(* Logix 5000 project; controller ODSI_Testing vendor 1 type 14 code 151 rev 20.19; software revision 20.05 *)

TASK MainTask (continuous, watchdog 500 ms) : MainProgram

MODULES
   Local : vendor 1 type 14 code 151 (Compact 0, rev 20.19)
      Expansion_Input_1 : 1769-IQ16 (Compact 4, rev 1.1, Input RPI 20 ms)   // Sink or Source
      Expansion_Input_2 : 1769-IQ32 (Compact 6, rev 3.1, Input RPI 20 ms)
      Discrete_IO : Embedded (Compact 1, rev 3.1, Output RPI 20 ms)
      Analog_IO : Embedded (Compact 2, rev 1.1, Output RPI 80 ms)
      Counters : Embedded (Compact 3, rev 1.1, Output RPI 20 ms)
      Expansion_Output_1 : vendor 1 type 7 code 75 (Compact 5, rev 1.1, Output RPI 20 ms)
END_MODULES

VAR_GLOBAL   (* controller tags *)
   B11_DELAY_ONS : BOOL;
   B12_DELAY_ONS : BOOL;
   B1_DELAY_ONS : BOOL;
   B9_DELAY_ONS : BOOL;
   DutyCycleOutput : BOOL := 1;   // 1.25 second duty cycle output
   DutyCycleTimer : TIMER := (PRE := 2500, ACC := 2111, EN := 1, TT := 1);   // Accumulates preset time then resets
   HMI_Stop_B1 : BOOL;   // Stop PB on HMI
   HMI_Stop_B11 : BOOL;   // Stop PB on HMI
   HMI_Stop_B12 : BOOL;   // Stop PB on HMI
   HMI_Stop_B9 : BOOL;   // Stop PB on HMI
   ODSI_Fail_Sample1_B1 : ALIAS FOR Local:4:I.Data.8;   // ODSI sent a fail signal for sample 1
   ODSI_Fail_Sample1_B11 : ALIAS FOR Local:1:I.Data.8;   // ODSI sent a fail signal for sample 1
   ODSI_Fail_Sample1_B12 : ALIAS FOR Local:6:I.Data.24;   // ODSI sent a fail signal for sample 1
   ODSI_Fail_Sample1_B9 : ALIAS FOR Local:6:I.Data.8;   // ODSI sent a fail signal for sample 1
   ODSI_Fail_Sample2_B1 : ALIAS FOR Local:4:I.Data.10;   // ODSI sent a fail signal for sample 2
   ODSI_Fail_Sample2_B11 : ALIAS FOR Local:1:I.Data.10;   // ODSI sent a fail signal for sample 2
   ODSI_Fail_Sample2_B12 : ALIAS FOR Local:6:I.Data.26;   // ODSI sent a fail signal for sample 2
   ODSI_Fail_Sample2_B9 : ALIAS FOR Local:6:I.Data.10;   // ODSI sent a fail signal for sample 2
   ODSI_Fail_Sample3_B1 : ALIAS FOR Local:4:I.Data.12;   // ODSI sent a fail signal for sample 3
   ODSI_Fail_Sample3_B11 : ALIAS FOR Local:1:I.Data.12;   // ODSI sent a fail signal for sample 3
   ODSI_Fail_Sample3_B12 : ALIAS FOR Local:6:I.Data.28;   // ODSI sent a fail signal for sample 3
   ODSI_Fail_Sample3_B9 : ALIAS FOR Local:6:I.Data.12;   // ODSI sent a fail signal for sample 3
   ODSI_Pass_Sample1_B1 : ALIAS FOR Local:4:I.Data.7;   // ODSI sent a pass signal for sample 1
   ODSI_Pass_Sample1_B11 : ALIAS FOR Local:1:I.Data.7;   // ODSI sent a pass signal for sample 1
   ODSI_Pass_Sample1_B12 : ALIAS FOR Local:6:I.Data.23;   // ODSI sent a pass signal for sample 1
   ODSI_Pass_Sample1_B9 : ALIAS FOR Local:6:I.Data.7;   // ODSI sent a pass signal for sample 1
   ODSI_Pass_Sample2_B1 : ALIAS FOR Local:4:I.Data.9;   // ODSI sent a pass signal for sample 2
   ODSI_Pass_Sample2_B11 : ALIAS FOR Local:1:I.Data.9;   // ODSI sent a pass signal for sample 2
   ODSI_Pass_Sample2_B12 : ALIAS FOR Local:6:I.Data.25;   // ODSI sent a pass signal for sample 2
   ODSI_Pass_Sample2_B9 : ALIAS FOR Local:6:I.Data.9;   // ODSI sent a pass signal for sample 2
   ODSI_Pass_Sample3_B1 : ALIAS FOR Local:4:I.Data.11;   // ODSI sent a pass signal for sample 3
   ODSI_Pass_Sample3_B11 : ALIAS FOR Local:1:I.Data.11;   // ODSI sent a pass signal for sample 3
   ODSI_Pass_Sample3_B12 : ALIAS FOR Local:6:I.Data.27;   // ODSI sent a pass signal for sample 3
   ODSI_Pass_Sample3_B9 : ALIAS FOR Local:6:I.Data.11;   // ODSI sent a pass signal for sample 3
   ODSI_Valve1_B1 : ALIAS FOR Local:4:I.Data.4;   // ODSI requests to open valve 1
   ODSI_Valve1_B11 : ALIAS FOR Local:1:I.Data.4;   // ODSI requests to open valve 1
   ODSI_Valve1_B12 : ALIAS FOR Local:6:I.Data.20;   // ODSI requests to open valve 1
   ODSI_Valve1_B9 : ALIAS FOR Local:6:I.Data.4;   // ODSI requests to open valve 1
   ODSI_Valve2_B1 : ALIAS FOR Local:4:I.Data.5;   // ODSI requests to open valve 2
   ODSI_Valve2_B11 : ALIAS FOR Local:1:I.Data.5;   // ODSI requests to open valve 2
   ODSI_Valve2_B12 : ALIAS FOR Local:6:I.Data.21;   // ODSI requests to open valve 2
   ODSI_Valve2_B9 : ALIAS FOR Local:6:I.Data.5;   // ODSI requests to open valve 2
   ODSI_Valve3_B1 : ALIAS FOR Local:4:I.Data.6;   // ODSI requests to open valve 3
   ODSI_Valve3_B11 : ALIAS FOR Local:1:I.Data.6;   // ODSI requests to open valve 3
   ODSI_Valve3_B12 : ALIAS FOR Local:6:I.Data.22;   // ODSI requests to open valve 3
   ODSI_Valve3_B9 : ALIAS FOR Local:6:I.Data.6;   // ODSI requests to open valve 3
   RandomDelay : DINT := 11;   // Random number generator 0-19
   RandomDelayDisplay_B1 : DINT;   // Snapshot of random delay at time of valve position request for B1
   RandomDelayDisplay_B11 : DINT;   // Snapshot of random delay at time of valve position request for B11
   RandomDelayDisplay_B12 : DINT;   // Snapshot of random delay at time of valve position request for B12
   RandomDelayDisplay_B9 : DINT;   // Snapshot of random delay at time of valve position request for B9
   RNG_Delay_Active_B1 : BOOL;   // HMI PB randomizing valve open delay
   RNG_Delay_Active_B11 : BOOL;   // HMI PB randomizing valve open delay
   RNG_Delay_Active_B12 : BOOL;   // HMI PB randomizing valve open delay
   RNG_Delay_Active_B9 : BOOL;   // HMI PB randomizing valve open delay
   S1_B11_10s_Timer : TIMER := (PRE := 10000);   // Releases "ACQC in" signal after 10 seconds
   S1_B12_10s_Timer : TIMER := (PRE := 10000);   // Releases "ACQC in" signal after 10 seconds
   S1_B1_10s_Timer : TIMER := (PRE := 10000);   // Releases "ACQC in" signal after 10 seconds
   S1_B9_10s_Timer : TIMER := (PRE := 10000);   // Releases "ACQC in" signal after 10 seconds
   S1_PB_Input_B1 : BOOL;   // HMI PB requesting sample 1
   S1_PB_Input_B11 : BOOL;   // HMI PB requesting sample 1
   S1_PB_Input_B12 : BOOL;   // HMI PB requesting sample 1
   S1_PB_Input_B9 : BOOL;   // HMI PB requesting sample 1
   S1_Request_B1 : ALIAS FOR Local:5:O.Data.0;   // Output to ODSI to request Sample 1
   S1_Request_B11 : ALIAS FOR Local:5:O.Data.16;   // Output to ODSI to request Sample 1
   S1_Request_B12 : ALIAS FOR Local:5:O.Data.24;   // Output to ODSI to request Sample 1
   S1_Request_B9 : ALIAS FOR Local:5:O.Data.8;   // Output to ODSI to request Sample 1
   S2_B11_10s_Timer : TIMER := (PRE := 10000);   // Releases "ACQC in" signal after 10 seconds
   S2_B12_10s_Timer : TIMER := (PRE := 10000);   // Releases "ACQC in" signal after 10 seconds
   S2_B1_10s_Timer : TIMER := (PRE := 10000);   // Releases "ACQC in" signal after 10 seconds
   S2_B9_10s_Timer : TIMER := (PRE := 10000);   // Releases "ACQC in" signal after 10 seconds
   S2_PB_Input_B1 : BOOL;   // HMI PB requesting sample 2
   S2_PB_Input_B11 : BOOL;   // HMI PB requesting sample 2
   S2_PB_Input_B12 : BOOL;   // HMI PB requesting sample 2
   S2_PB_Input_B9 : BOOL;   // HMI PB requesting sample 2
   S2_Request_B1 : ALIAS FOR Local:5:O.Data.1;   // Output to ODSI to request Sample 2
   S2_Request_B11 : ALIAS FOR Local:5:O.Data.17;   // Output to ODSI to request Sample 2
   S2_Request_B12 : ALIAS FOR Local:5:O.Data.25;   // Output to ODSI to request Sample 2
   S2_Request_B9 : ALIAS FOR Local:5:O.Data.9;   // Output to ODSI to request Sample 2
   S3_B11_10s_Timer : TIMER := (PRE := 10000);   // Releases "ACQC in" signal after 10 seconds
   S3_B12_10s_Timer : TIMER := (PRE := 10000);   // Releases "ACQC in" signal after 10 seconds
   S3_B1_10s_Timer : TIMER := (PRE := 10000);   // Releases "ACQC in" signal after 10 seconds
   S3_B9_10s_Timer : TIMER := (PRE := 10000);   // Releases "ACQC in" signal after 10 seconds
   S3_PB_Input_B1 : BOOL;   // HMI PB requesting sample 3
   S3_PB_Input_B11 : BOOL;   // HMI PB requesting sample 3
   S3_PB_Input_B12 : BOOL;   // HMI PB requesting sample 3
   S3_PB_Input_B9 : BOOL;   // HMI PB requesting sample 3
   S3_Request_B1 : ALIAS FOR Local:5:O.Data.2;   // Output to ODSI to request Sample 3
   S3_Request_B11 : ALIAS FOR Local:5:O.Data.18;   // Output to ODSI to request Sample 3
   S3_Request_B12 : ALIAS FOR Local:5:O.Data.26;   // Output to ODSI to request Sample 3
   S3_Request_B9 : ALIAS FOR Local:5:O.Data.10;   // Output to ODSI to request Sample 3
   System_Running_B1 : ALIAS FOR Local:4:I.Data.3;   // ODSI signal that indicates the system is currently analyzing a sample
   System_Running_B11 : ALIAS FOR Local:1:I.Data.3;   // ODSI signal that indicates the system is currently analyzing a sample
   System_Running_B12 : ALIAS FOR Local:6:I.Data.19;   // ODSI signal that indicates the system is currently analyzing a sample
   System_Running_B9 : ALIAS FOR Local:6:I.Data.3;   // ODSI signal that indicates the system is currently analyzing a sample
   SystemTime : DINT[7] := ([0] := 1998, [1] := 1, [2] := 22, [3] := 5, [4] := 42, [5] := 32, [6] := 563285);
        [1]   // Month
        [4]   // Minute
        [0]   // Year
        [2]   // Day
        [3]   // Hour
        [5]   // Second
        [6]   // Microsecond
   Temp : DINT := 10;
   Valve1_Open_B1 : ALIAS FOR Local:5:O.Data.3;   // Output to ODSI confirming valve 1 is open
   Valve1_Open_B11 : ALIAS FOR Local:5:O.Data.19;   // Output to ODSI confirming valve 1 is open
   Valve1_Open_B12 : ALIAS FOR Local:5:O.Data.27;   // Output to ODSI confirming valve 1 is open
   Valve1_Open_B9 : ALIAS FOR Local:5:O.Data.11;   // Output to ODSI confirming valve 1 is open
   Valve1_Open_Delay_B1 : TIMER;   // Delay after Request is Initiated from ODSI
   Valve1_Open_Delay_B11 : TIMER;   // Delay after Request is Initiated from ODSI
   Valve1_Open_Delay_B12 : TIMER;   // Delay after Request is Initiated from ODSI
   Valve1_Open_Delay_B9 : TIMER;   // Delay after Request is Initiated from ODSI
   Valve1_Open_Random_Delay_B1 : TIMER := (PRE := 11000);   // Randomized delay after request for valve position is received from ODSI
   Valve1_Open_Random_Delay_B11 : TIMER := (PRE := 11000);   // Randomized delay after request for valve position is received from ODSI
   Valve1_Open_Random_Delay_B12 : TIMER := (PRE := 11000);   // Randomized delay after request for valve position is received from ODSI
   Valve1_Open_Random_Delay_B9 : TIMER := (PRE := 11000);   // Randomized delay after request for valve position is received from ODSI
   Valve2_Open_B1 : ALIAS FOR Local:5:O.Data.4;   // Output to ODSI confirming valve 2 is open
   Valve2_Open_B11 : ALIAS FOR Local:5:O.Data.20;   // Output to ODSI confirming valve 2 is open
   Valve2_Open_B12 : ALIAS FOR Local:5:O.Data.28;   // Output to ODSI confirming valve 2 is open
   Valve2_Open_B9 : ALIAS FOR Local:5:O.Data.12;   // Output to ODSI confirming valve 2 is open
   Valve2_Open_Delay_B1 : TIMER;   // Delay after Request is Initiated from ODSI
   Valve2_Open_Delay_B11 : TIMER;   // Delay after Request is Initiated from ODSI
   Valve2_Open_Delay_B12 : TIMER;   // Delay after Request is Initiated from ODSI
   Valve2_Open_Delay_B9 : TIMER;   // Delay after Request is Initiated from ODSI
   Valve2_Open_Random_Delay_B1 : TIMER := (PRE := 11000);   // Randomized delay after request for valve position is received from ODSI
   Valve2_Open_Random_Delay_B11 : TIMER := (PRE := 11000);   // Randomized delay after request for valve position is received from ODSI
   Valve2_Open_Random_Delay_B12 : TIMER := (PRE := 11000);   // Randomized delay after request for valve position is received from ODSI
   Valve2_Open_Random_Delay_B9 : TIMER := (PRE := 11000);   // Randomized delay after request for valve position is received from ODSI
   Valve3_Open_B1 : ALIAS FOR Local:5:O.Data.5;   // Output to ODSI confirming valve 3 is open
   Valve3_Open_B11 : ALIAS FOR Local:5:O.Data.21;   // Output to ODSI confirming valve 3 is open
   Valve3_Open_B12 : ALIAS FOR Local:5:O.Data.29;   // Output to ODSI confirming valve 3 is open
   Valve3_Open_B9 : ALIAS FOR Local:5:O.Data.13;   // Output to ODSI confirming valve 3 is open
   Valve3_Open_Delay_B1 : TIMER;   // Delay after Request is Initiated from ODSI
   Valve3_Open_Delay_B11 : TIMER;   // Delay after Request is Initiated from ODSI
   Valve3_Open_Delay_B12 : TIMER;   // Delay after Request is Initiated from ODSI
   Valve3_Open_Delay_B9 : TIMER;   // Delay after Request is Initiated from ODSI
   Valve3_Open_Random_Delay_B1 : TIMER := (PRE := 11000);   // Randomized delay after request for valve position is received from ODSI
   Valve3_Open_Random_Delay_B11 : TIMER := (PRE := 11000);   // Randomized delay after request for valve position is received from ODSI
   Valve3_Open_Random_Delay_B12 : TIMER := (PRE := 11000);   // Randomized delay after request for valve position is received from ODSI
   Valve3_Open_Random_Delay_B9 : TIMER := (PRE := 11000);   // Randomized delay after request for valve position is received from ODSI
   Valve_Block_B1 : BOOL;   // HMI PB to prevent valves from opening
   Valve_Block_B11 : BOOL;   // HMI PB to prevent valves from opening
   Valve_Block_B12 : BOOL;   // HMI PB to prevent valves from opening
   Valve_Block_B9 : BOOL;   // HMI PB to prevent valves from opening
   Valve_Delay_B1 : DINT;
   Valve_Delay_B11 : DINT;
   Valve_Delay_B12 : DINT;
   Valve_Delay_B9 : DINT;
END_VAR

PROGRAM MainProgram   (* main routine MainRoutine *)

ROUTINE MainRoutine   (* ladder *)
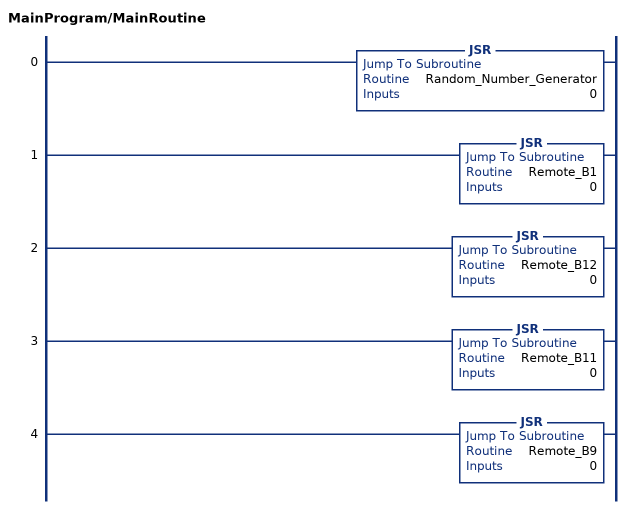
   0: JSR(Random_Number_Generator,0);
   1: JSR(Remote_B1,0);
   2: JSR(Remote_B12,0);
   3: JSR(Remote_B11,0);
   4: JSR(Remote_B9,0);
END_ROUTINE

ROUTINE Random_Number_Generator   (* ladder *)
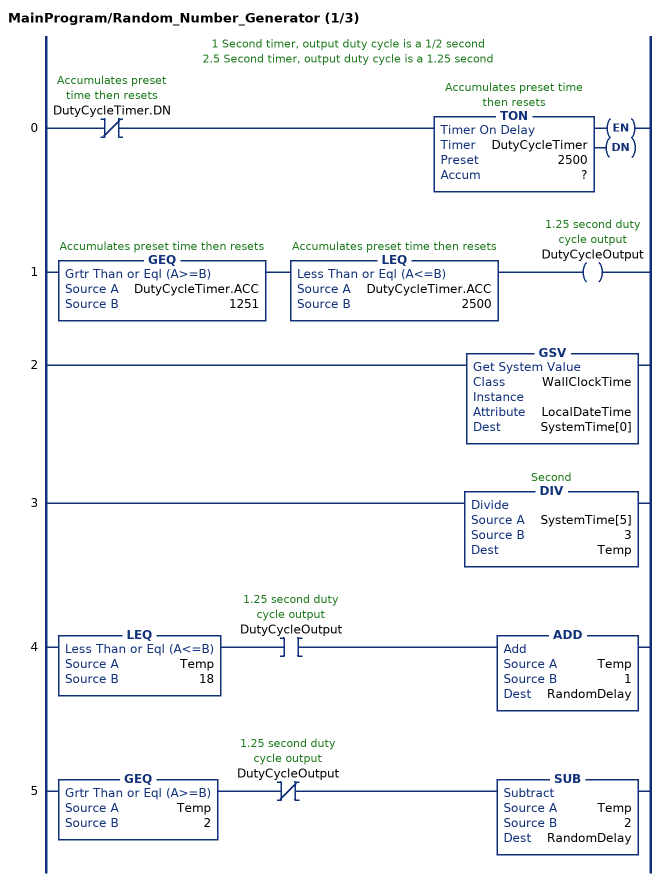
   // 1 Second timer, output duty cycle is a 1/2 second
   // 2.5 Second timer, output duty cycle is a 1.25 second
   0: XIO(DutyCycleTimer.DN)TON(DutyCycleTimer,?,?);
   1: GEQ(DutyCycleTimer.ACC,1251)LEQ(DutyCycleTimer.ACC,2500)OTE(DutyCycleOutput);
   2: GSV(WallClockTime,,LocalDateTime,SystemTime[0]);
   3: DIV(SystemTime[5],3,Temp);
   4: LEQ(Temp,18)XIC(DutyCycleOutput)ADD(Temp,1,RandomDelay);
   5: GEQ(Temp,2)XIO(DutyCycleOutput)SUB(Temp,2,RandomDelay);
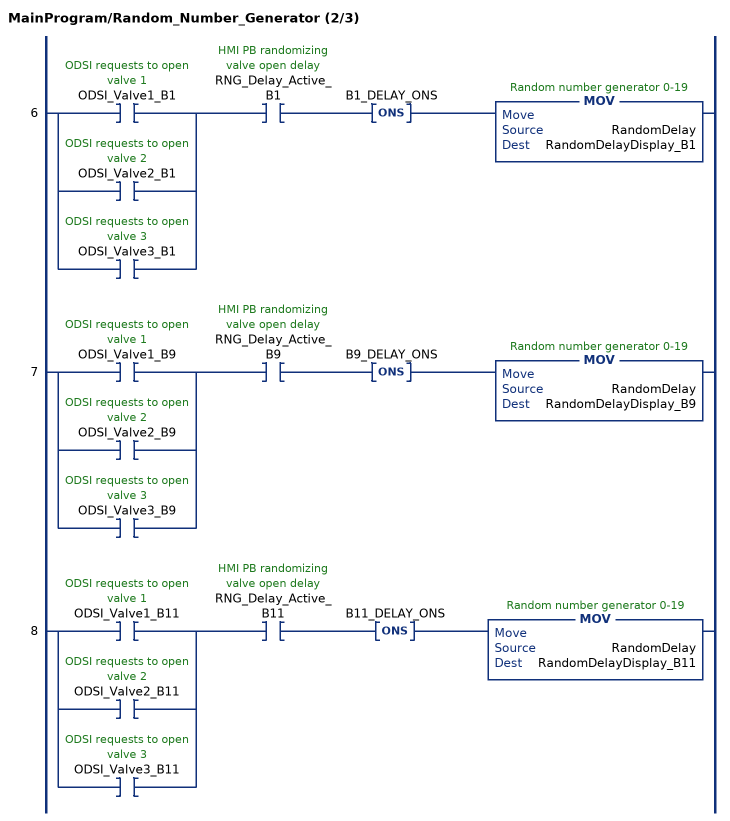
   6: [XIC(ODSI_Valve1_B1) ,XIC(ODSI_Valve2_B1) ,XIC(ODSI_Valve3_B1) ]XIC(RNG_Delay_Active_B1)ONS(B1_DELAY_ONS)MOV(RandomDelay,RandomDelayDisplay_B1);
   7: [XIC(ODSI_Valve1_B9) ,XIC(ODSI_Valve2_B9) ,XIC(ODSI_Valve3_B9) ]XIC(RNG_Delay_Active_B9)ONS(B9_DELAY_ONS)MOV(RandomDelay,RandomDelayDisplay_B9);
   8: [XIC(ODSI_Valve1_B11) ,XIC(ODSI_Valve2_B11) ,XIC(ODSI_Valve3_B11) ]XIC(RNG_Delay_Active_B11)ONS(B11_DELAY_ONS)MOV(RandomDelay,RandomDelayDisplay_B11);
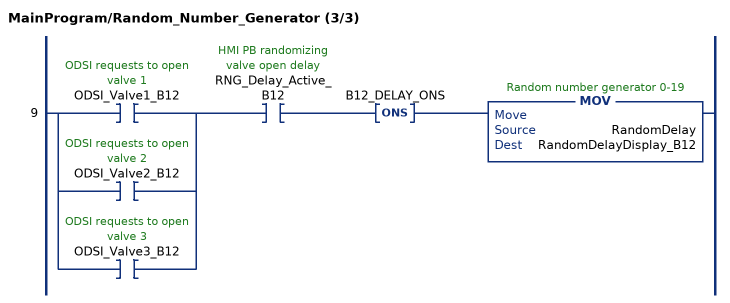
   9: [XIC(ODSI_Valve1_B12) ,XIC(ODSI_Valve2_B12) ,XIC(ODSI_Valve3_B12) ]XIC(RNG_Delay_Active_B12)ONS(B12_DELAY_ONS)MOV(RandomDelay,RandomDelayDisplay_B12);
END_ROUTINE

ROUTINE Remote_B1   (* ladder *)
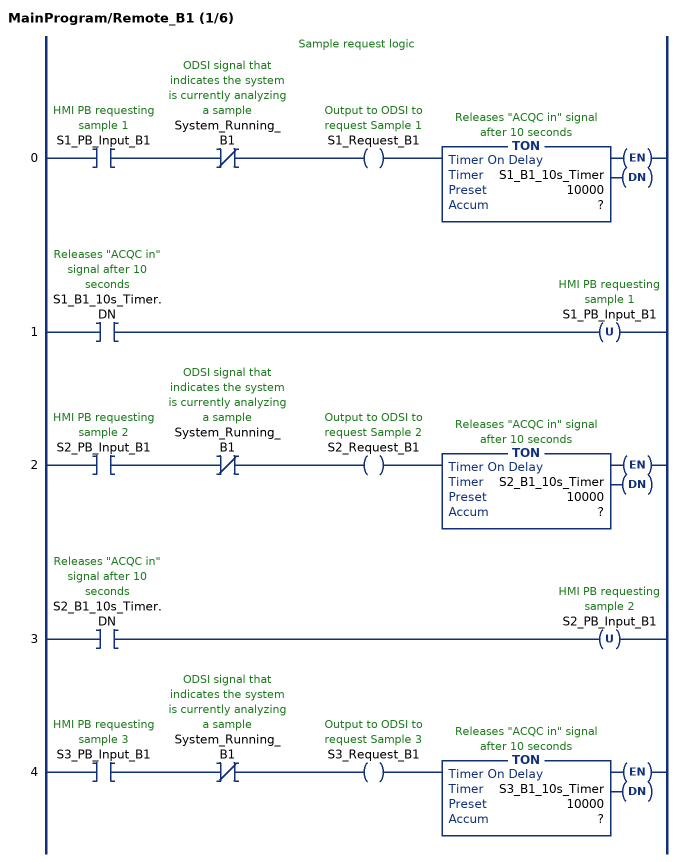
   // Sample request logic
   0: XIC(S1_PB_Input_B1)XIO(System_Running_B1)OTE(S1_Request_B1)TON(S1_B1_10s_Timer,?,?);
   1: XIC(S1_B1_10s_Timer.DN)OTU(S1_PB_Input_B1);
   2: XIC(S2_PB_Input_B1)XIO(System_Running_B1)OTE(S2_Request_B1)TON(S2_B1_10s_Timer,?,?);
   3: XIC(S2_B1_10s_Timer.DN)OTU(S2_PB_Input_B1);
   4: XIC(S3_PB_Input_B1)XIO(System_Running_B1)OTE(S3_Request_B1)TON(S3_B1_10s_Timer,?,?);
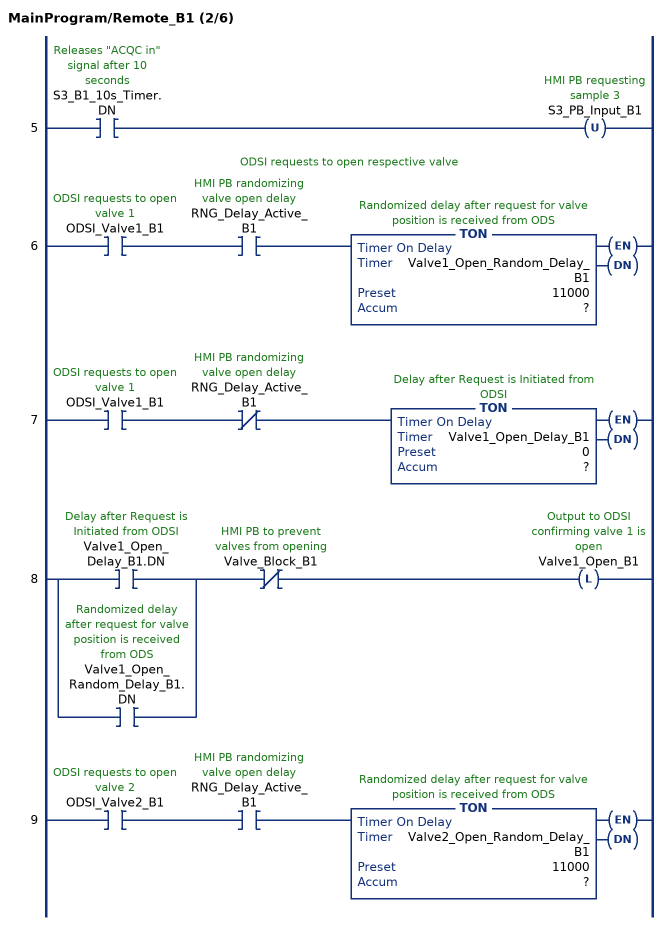
   5: XIC(S3_B1_10s_Timer.DN)OTU(S3_PB_Input_B1);
   // ODSI requests to open respective valve
   6: XIC(ODSI_Valve1_B1)XIC(RNG_Delay_Active_B1)TON(Valve1_Open_Random_Delay_B1,?,?);
   7: XIC(ODSI_Valve1_B1)XIO(RNG_Delay_Active_B1)TON(Valve1_Open_Delay_B1,?,?);
   8: [XIC(Valve1_Open_Delay_B1.DN) ,XIC(Valve1_Open_Random_Delay_B1.DN) ]XIO(Valve_Block_B1)OTL(Valve1_Open_B1);
   9: XIC(ODSI_Valve2_B1)XIC(RNG_Delay_Active_B1)TON(Valve2_Open_Random_Delay_B1,?,?);
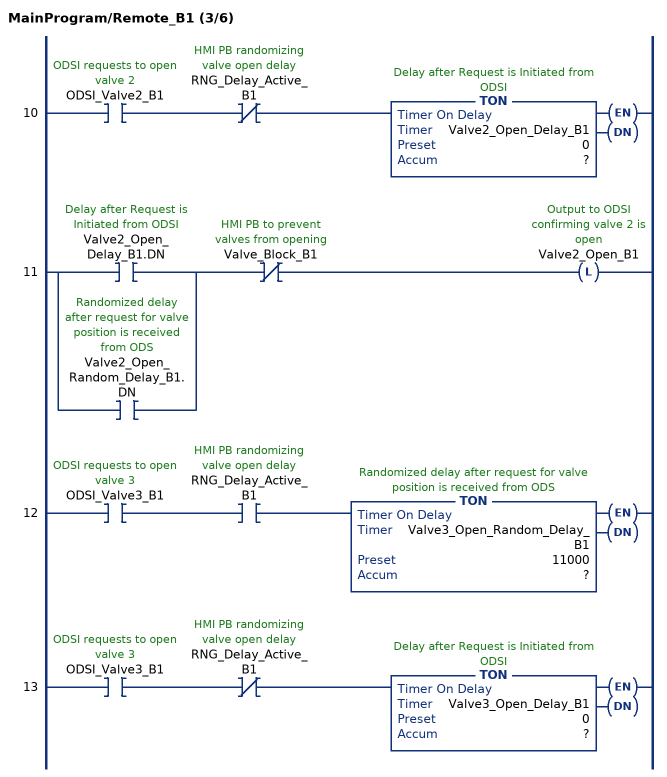
   10: XIC(ODSI_Valve2_B1)XIO(RNG_Delay_Active_B1)TON(Valve2_Open_Delay_B1,?,?);
   11: [XIC(Valve2_Open_Delay_B1.DN) ,XIC(Valve2_Open_Random_Delay_B1.DN) ]XIO(Valve_Block_B1)OTL(Valve2_Open_B1);
   12: XIC(ODSI_Valve3_B1)XIC(RNG_Delay_Active_B1)TON(Valve3_Open_Random_Delay_B1,?,?);
   13: XIC(ODSI_Valve3_B1)XIO(RNG_Delay_Active_B1)TON(Valve3_Open_Delay_B1,?,?);
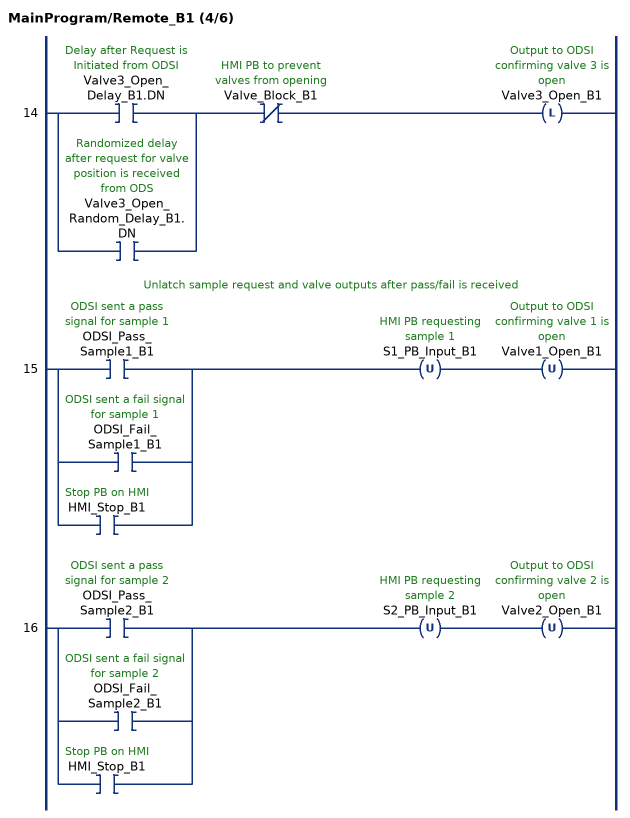
   14: [XIC(Valve3_Open_Delay_B1.DN) ,XIC(Valve3_Open_Random_Delay_B1.DN) ]XIO(Valve_Block_B1)OTL(Valve3_Open_B1);
   // Unlatch sample request and valve outputs after pass/fail is received
   15: [XIC(ODSI_Pass_Sample1_B1) ,XIC(ODSI_Fail_Sample1_B1) ,XIC(HMI_Stop_B1) ]OTU(S1_PB_Input_B1)OTU(Valve1_Open_B1);
   16: [XIC(ODSI_Pass_Sample2_B1) ,XIC(ODSI_Fail_Sample2_B1) ,XIC(HMI_Stop_B1) ]OTU(S2_PB_Input_B1)OTU(Valve2_Open_B1);
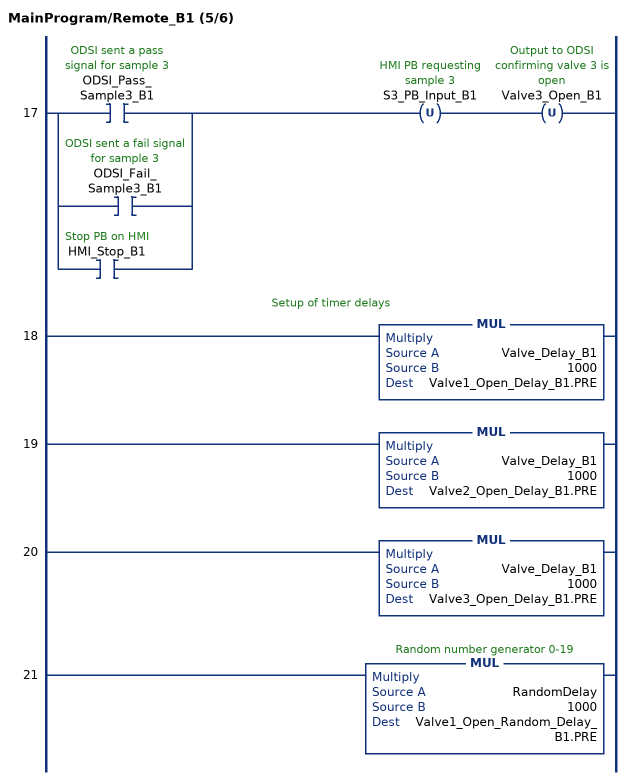
   17: [XIC(ODSI_Pass_Sample3_B1) ,XIC(ODSI_Fail_Sample3_B1) ,XIC(HMI_Stop_B1) ]OTU(S3_PB_Input_B1)OTU(Valve3_Open_B1);
   // Setup of timer delays
   18: MUL(Valve_Delay_B1,1000,Valve1_Open_Delay_B1.PRE);
   19: MUL(Valve_Delay_B1,1000,Valve2_Open_Delay_B1.PRE);
   20: MUL(Valve_Delay_B1,1000,Valve3_Open_Delay_B1.PRE);
   21: MUL(RandomDelay,1000,Valve1_Open_Random_Delay_B1.PRE);
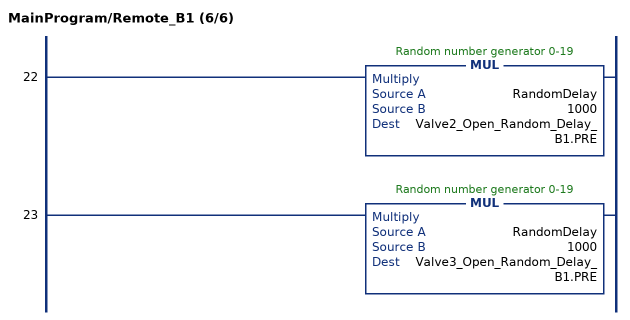
   22: MUL(RandomDelay,1000,Valve2_Open_Random_Delay_B1.PRE);
   23: MUL(RandomDelay,1000,Valve3_Open_Random_Delay_B1.PRE);
END_ROUTINE

ROUTINE Remote_B11   (* ladder *)
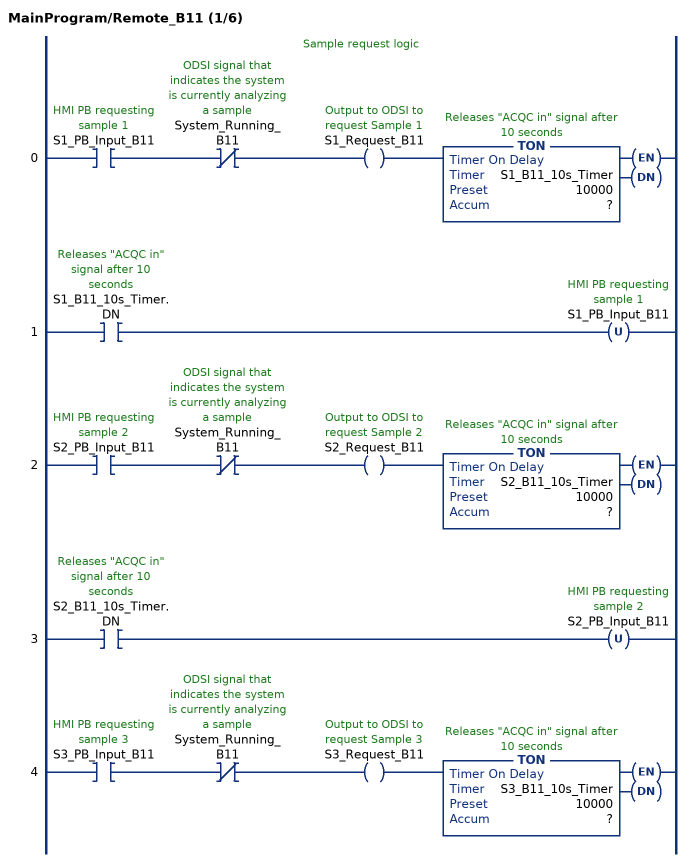
   // Sample request logic
   0: XIC(S1_PB_Input_B11)XIO(System_Running_B11)OTE(S1_Request_B11)TON(S1_B11_10s_Timer,?,?);
   1: XIC(S1_B11_10s_Timer.DN)OTU(S1_PB_Input_B11);
   2: XIC(S2_PB_Input_B11)XIO(System_Running_B11)OTE(S2_Request_B11)TON(S2_B11_10s_Timer,?,?);
   3: XIC(S2_B11_10s_Timer.DN)OTU(S2_PB_Input_B11);
   4: XIC(S3_PB_Input_B11)XIO(System_Running_B11)OTE(S3_Request_B11)TON(S3_B11_10s_Timer,?,?);
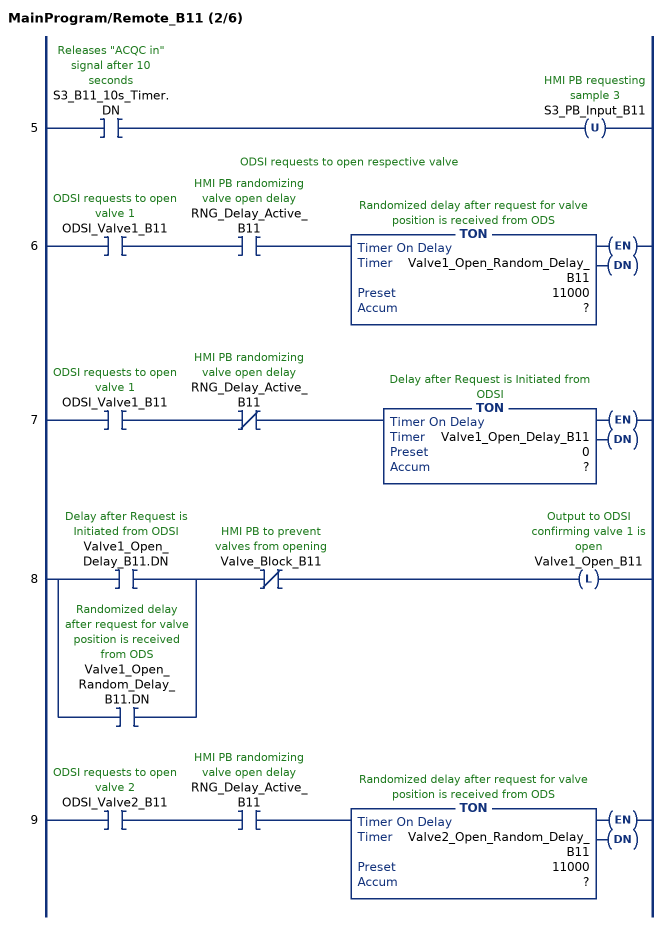
   5: XIC(S3_B11_10s_Timer.DN)OTU(S3_PB_Input_B11);
   // ODSI requests to open respective valve
   6: XIC(ODSI_Valve1_B11)XIC(RNG_Delay_Active_B11)TON(Valve1_Open_Random_Delay_B11,?,?);
   7: XIC(ODSI_Valve1_B11)XIO(RNG_Delay_Active_B11)TON(Valve1_Open_Delay_B11,?,?);
   8: [XIC(Valve1_Open_Delay_B11.DN) ,XIC(Valve1_Open_Random_Delay_B11.DN) ]XIO(Valve_Block_B11)OTL(Valve1_Open_B11);
   9: XIC(ODSI_Valve2_B11)XIC(RNG_Delay_Active_B11)TON(Valve2_Open_Random_Delay_B11,?,?);
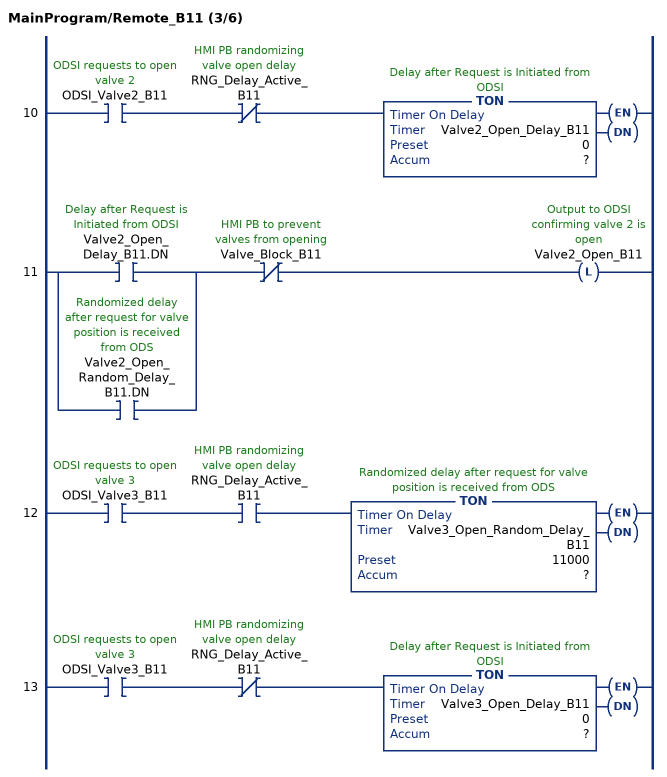
   10: XIC(ODSI_Valve2_B11)XIO(RNG_Delay_Active_B11)TON(Valve2_Open_Delay_B11,?,?);
   11: [XIC(Valve2_Open_Delay_B11.DN) ,XIC(Valve2_Open_Random_Delay_B11.DN) ]XIO(Valve_Block_B11)OTL(Valve2_Open_B11);
   12: XIC(ODSI_Valve3_B11)XIC(RNG_Delay_Active_B11)TON(Valve3_Open_Random_Delay_B11,?,?);
   13: XIC(ODSI_Valve3_B11)XIO(RNG_Delay_Active_B11)TON(Valve3_Open_Delay_B11,?,?);
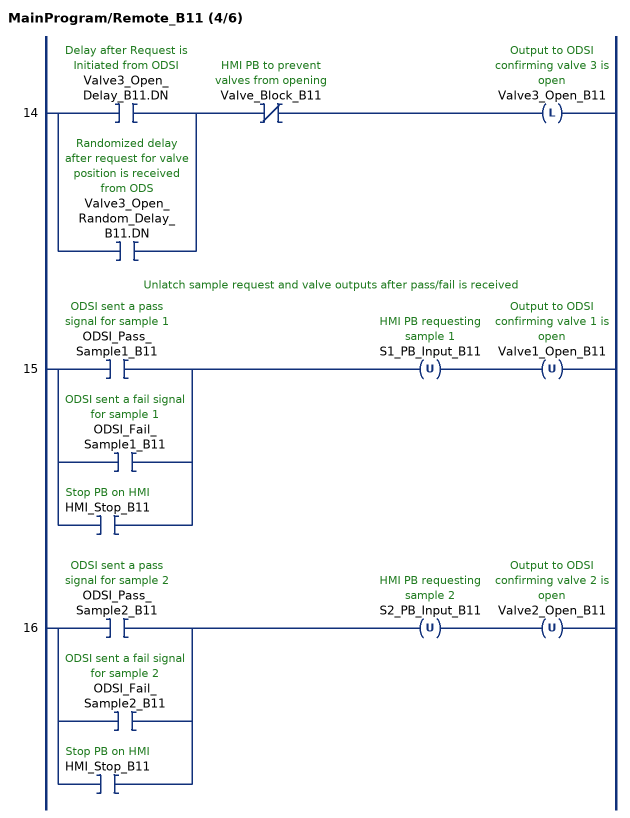
   14: [XIC(Valve3_Open_Delay_B11.DN) ,XIC(Valve3_Open_Random_Delay_B11.DN) ]XIO(Valve_Block_B11)OTL(Valve3_Open_B11);
   // Unlatch sample request and valve outputs after pass/fail is received
   15: [XIC(ODSI_Pass_Sample1_B11) ,XIC(ODSI_Fail_Sample1_B11) ,XIC(HMI_Stop_B11) ]OTU(S1_PB_Input_B11)OTU(Valve1_Open_B11);
   16: [XIC(ODSI_Pass_Sample2_B11) ,XIC(ODSI_Fail_Sample2_B11) ,XIC(HMI_Stop_B11) ]OTU(S2_PB_Input_B11)OTU(Valve2_Open_B11);
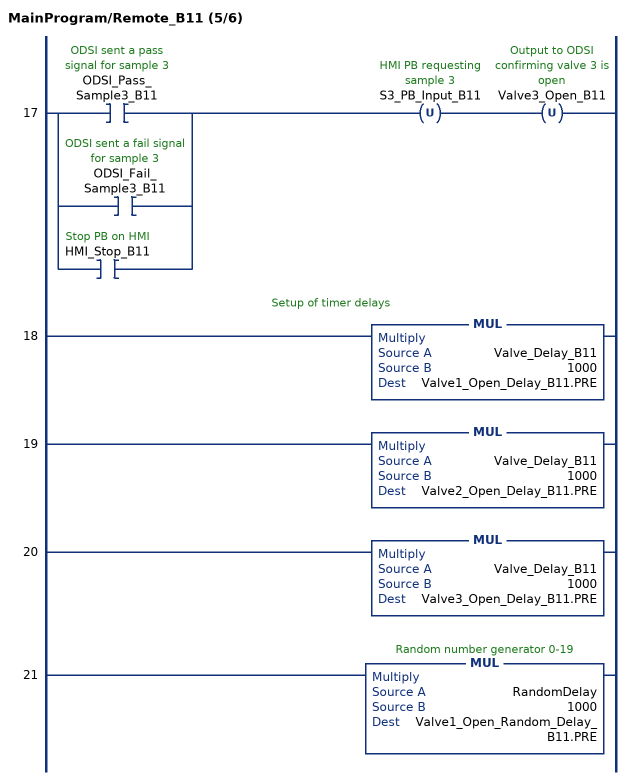
   17: [XIC(ODSI_Pass_Sample3_B11) ,XIC(ODSI_Fail_Sample3_B11) ,XIC(HMI_Stop_B11) ]OTU(S3_PB_Input_B11)OTU(Valve3_Open_B11);
   // Setup of timer delays
   18: MUL(Valve_Delay_B11,1000,Valve1_Open_Delay_B11.PRE);
   19: MUL(Valve_Delay_B11,1000,Valve2_Open_Delay_B11.PRE);
   20: MUL(Valve_Delay_B11,1000,Valve3_Open_Delay_B11.PRE);
   21: MUL(RandomDelay,1000,Valve1_Open_Random_Delay_B11.PRE);
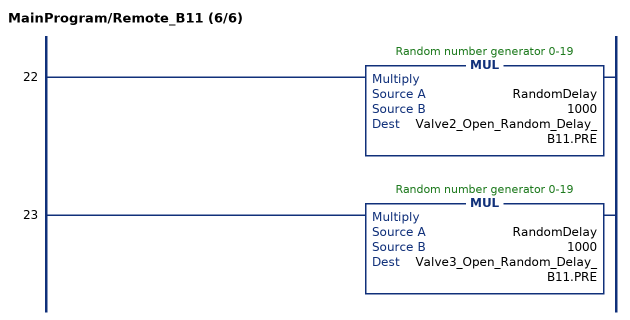
   22: MUL(RandomDelay,1000,Valve2_Open_Random_Delay_B11.PRE);
   23: MUL(RandomDelay,1000,Valve3_Open_Random_Delay_B11.PRE);
END_ROUTINE

ROUTINE Remote_B12   (* ladder *)
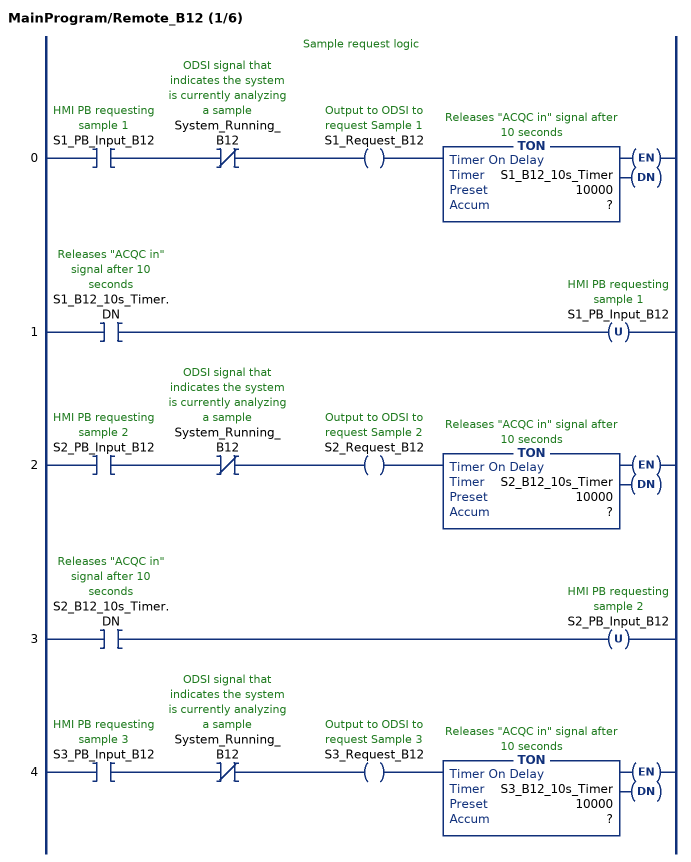
   // Sample request logic
   0: XIC(S1_PB_Input_B12)XIO(System_Running_B12)OTE(S1_Request_B12)TON(S1_B12_10s_Timer,?,?);
   1: XIC(S1_B12_10s_Timer.DN)OTU(S1_PB_Input_B12);
   2: XIC(S2_PB_Input_B12)XIO(System_Running_B12)OTE(S2_Request_B12)TON(S2_B12_10s_Timer,?,?);
   3: XIC(S2_B12_10s_Timer.DN)OTU(S2_PB_Input_B12);
   4: XIC(S3_PB_Input_B12)XIO(System_Running_B12)OTE(S3_Request_B12)TON(S3_B12_10s_Timer,?,?);
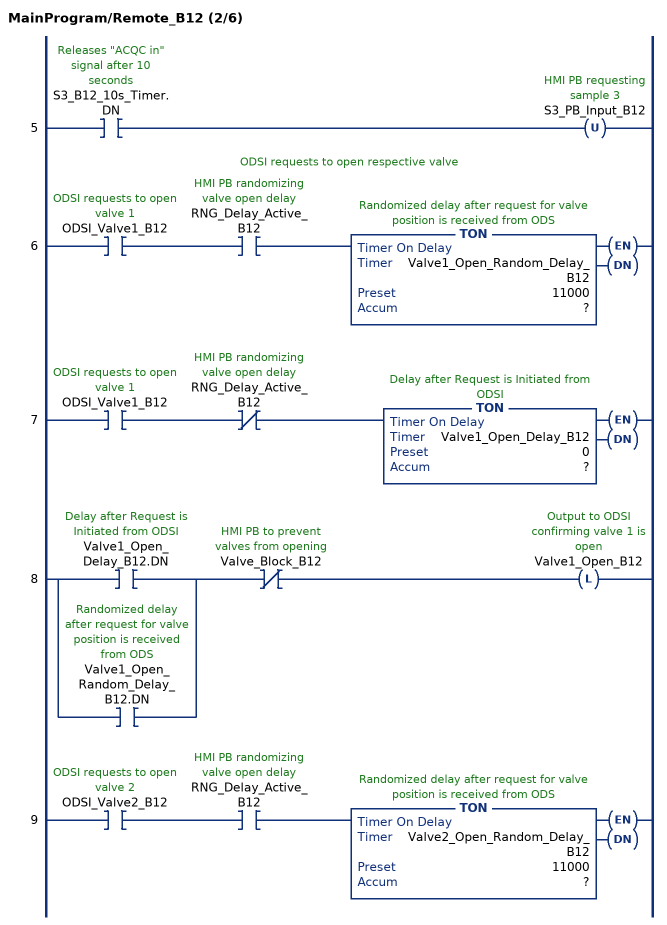
   5: XIC(S3_B12_10s_Timer.DN)OTU(S3_PB_Input_B12);
   // ODSI requests to open respective valve
   6: XIC(ODSI_Valve1_B12)XIC(RNG_Delay_Active_B12)TON(Valve1_Open_Random_Delay_B12,?,?);
   7: XIC(ODSI_Valve1_B12)XIO(RNG_Delay_Active_B12)TON(Valve1_Open_Delay_B12,?,?);
   8: [XIC(Valve1_Open_Delay_B12.DN) ,XIC(Valve1_Open_Random_Delay_B12.DN) ]XIO(Valve_Block_B12)OTL(Valve1_Open_B12);
   9: XIC(ODSI_Valve2_B12)XIC(RNG_Delay_Active_B12)TON(Valve2_Open_Random_Delay_B12,?,?);
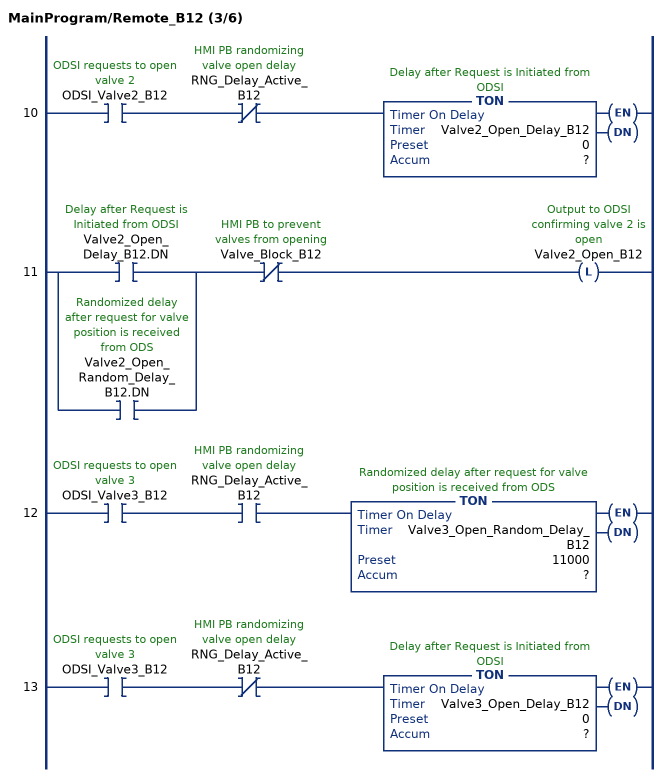
   10: XIC(ODSI_Valve2_B12)XIO(RNG_Delay_Active_B12)TON(Valve2_Open_Delay_B12,?,?);
   11: [XIC(Valve2_Open_Delay_B12.DN) ,XIC(Valve2_Open_Random_Delay_B12.DN) ]XIO(Valve_Block_B12)OTL(Valve2_Open_B12);
   12: XIC(ODSI_Valve3_B12)XIC(RNG_Delay_Active_B12)TON(Valve3_Open_Random_Delay_B12,?,?);
   13: XIC(ODSI_Valve3_B12)XIO(RNG_Delay_Active_B12)TON(Valve3_Open_Delay_B12,?,?);
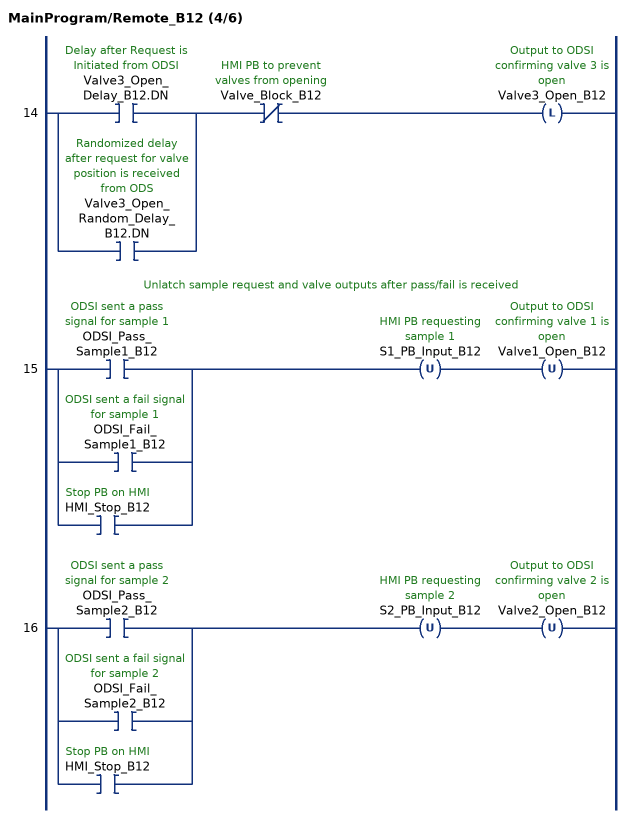
   14: [XIC(Valve3_Open_Delay_B12.DN) ,XIC(Valve3_Open_Random_Delay_B12.DN) ]XIO(Valve_Block_B12)OTL(Valve3_Open_B12);
   // Unlatch sample request and valve outputs after pass/fail is received
   15: [XIC(ODSI_Pass_Sample1_B12) ,XIC(ODSI_Fail_Sample1_B12) ,XIC(HMI_Stop_B12) ]OTU(S1_PB_Input_B12)OTU(Valve1_Open_B12);
   16: [XIC(ODSI_Pass_Sample2_B12) ,XIC(ODSI_Fail_Sample2_B12) ,XIC(HMI_Stop_B12) ]OTU(S2_PB_Input_B12)OTU(Valve2_Open_B12);
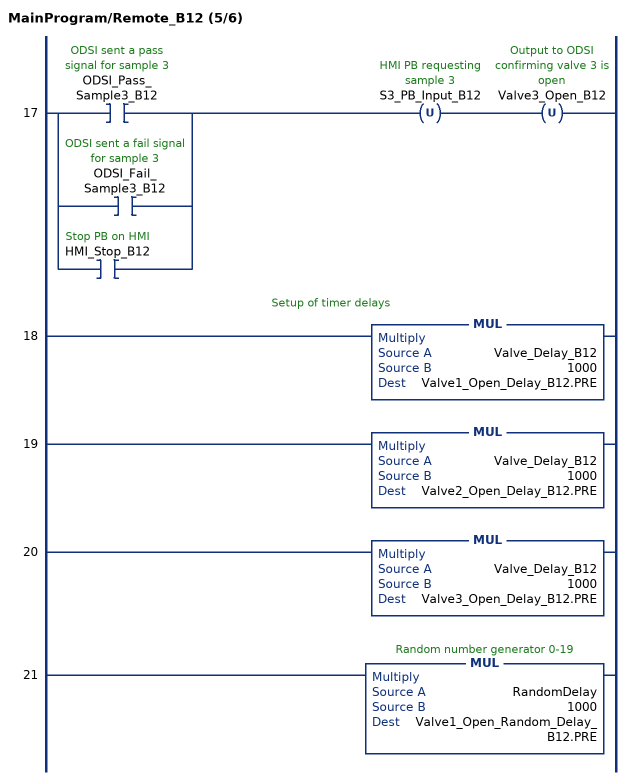
   17: [XIC(ODSI_Pass_Sample3_B12) ,XIC(ODSI_Fail_Sample3_B12) ,XIC(HMI_Stop_B12) ]OTU(S3_PB_Input_B12)OTU(Valve3_Open_B12);
   // Setup of timer delays
   18: MUL(Valve_Delay_B12,1000,Valve1_Open_Delay_B12.PRE);
   19: MUL(Valve_Delay_B12,1000,Valve2_Open_Delay_B12.PRE);
   20: MUL(Valve_Delay_B12,1000,Valve3_Open_Delay_B12.PRE);
   21: MUL(RandomDelay,1000,Valve1_Open_Random_Delay_B12.PRE);
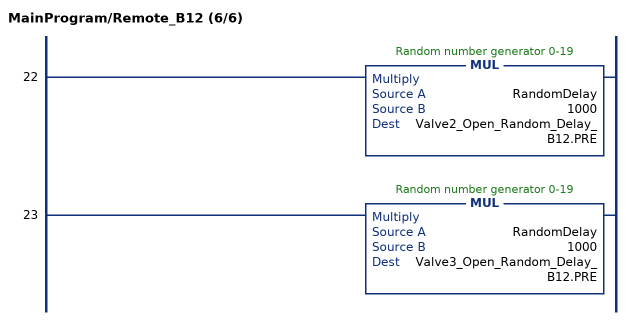
   22: MUL(RandomDelay,1000,Valve2_Open_Random_Delay_B12.PRE);
   23: MUL(RandomDelay,1000,Valve3_Open_Random_Delay_B12.PRE);
END_ROUTINE
